(* IEC 61131-3 sources: moqui-plc/iec61131/moqui/framework/src/main/org/moqui/context, 20 files *)

(* ---- LogCmd.dut ---- *)
(*#-#-#-#-#-#-#-#-#-#---Declaration---#-#-#-#-#-#-#-#-#-#-#-#-#*)

{attribute 'qualified_only'}
TYPE LogCmd : (
    Idle := 0, (* Waiting for commands *)
    Push, (* Inserting a new log entry *)
	IncrementLast, (* Update the last log entry *)
	Peek, (* Read a log entry without removing it *)
	Pop, (* It actually removes the appended log entries *)
    Clear (* Complete buffer reset *)
); END_TYPE

(* ---- LogCmd.st ---- *)
TYPE LogCmd : (
    Idle := 0, (* Waiting for commands *)
    Push, (* Inserting a new log entry *)
	IncrementLast, (* Update the last log entry *)
	Peek, (* Read a log entry without removing it *)
	Pop, (* It actually removes the appended log entries *)
    Clear (* Complete buffer reset *)
); END_TYPE

(* ---- LogEvent.dut ---- *)
(*#-#-#-#-#-#-#-#-#-#---Declaration---#-#-#-#-#-#-#-#-#-#-#-#-#*)

TYPE LogEvent : STRUCT
	(* Unique identifier for the log event *)
    logEventId : STRING;
    loggerName : STRING;
	marker : LogMarker;
    level : LogLevel;
    logEventDate : DATE_AND_TIME;
	source : STRING;
	payloadType : LogPayloadType;
    payload : LogPayload;
	(* contextData: STRING; *)
	(* Number of times this log event was repeated, for compression *)
    repeatCount : UINT;
END_STRUCT END_TYPE

(* ---- LogEvent.st ---- *)
TYPE LogEvent : STRUCT
	(* Unique identifier for the log event *)
    logEventId : STRING;
    loggerName : STRING;
	marker : LogMarker;
    level : LogLevel;
    logEventDate : DATE_AND_TIME;
	source : STRING;
	payloadType : LogPayloadType;
    payload : LogPayload;
	(* contextData: STRING; *)
	(* Number of times this log event was repeated, for compression *)
    repeatCount : UINT;
END_STRUCT END_TYPE

(* ---- LogLevel.dut ---- *)
(*#-#-#-#-#-#-#-#-#-#---Declaration---#-#-#-#-#-#-#-#-#-#-#-#-#*)

{attribute 'qualified_only'}
TYPE LogLevel : (
	Trace := 0,
	Debug,
	Info,
	Warn,
	Error,
	Fatal,
	All,
	Off
); END_TYPE

(* ---- LogLevel.st ---- *)
TYPE LogLevel : (
	Trace := 0,
	Debug,
	Info,
	Warn,
	Error,
	Fatal,
	All,
	Off
); END_TYPE

(* ---- LogMarker.dut ---- *)
(*#-#-#-#-#-#-#-#-#-#---Declaration---#-#-#-#-#-#-#-#-#-#-#-#-#*)

{attribute 'qualified_only'}
{attribute 'strict'}
TYPE LogMarker : (
	Diagnostics := 0,
	Lifecycle,
	Integration,
	Health,
	Telemetry,
	AuditLog,
	Kpi,
	Measurement
); END_TYPE

(* ---- LogMarker.st ---- *)
TYPE LogMarker : (
	Diagnostics := 0,
	Lifecycle,
	Integration,
	Health,
	Telemetry,
	AuditLog,
	Kpi,
	Measurement
); END_TYPE

(* ---- LogPayload.dut ---- *)
(*#-#-#-#-#-#-#-#-#-#---Declaration---#-#-#-#-#-#-#-#-#-#-#-#-#*)

TYPE LogPayload : UNION
	message : STRING;
    enumValue : UINT;
    numericValue : LREAL;
END_UNION END_TYPE

(* ---- LogPayload.st ---- *)
TYPE LogPayload : UNION
	message : STRING;
    enumValue : UINT;
    numericValue : LREAL;
END_UNION END_TYPE

(* ---- LogPayloadType.dut ---- *)
(*#-#-#-#-#-#-#-#-#-#---Declaration---#-#-#-#-#-#-#-#-#-#-#-#-#*)

{attribute 'qualified_only'}
TYPE LogPayloadType : (
    Text := 0,
	Numeric,
	Enum
); END_TYPE

(* ---- LogPayloadType.st ---- *)
TYPE LogPayloadType : (
    Text := 0,
	Numeric,
	Enum
); END_TYPE

(* ---- LogSource.dut ---- *)
(*#-#-#-#-#-#-#-#-#-#---Declaration---#-#-#-#-#-#-#-#-#-#-#-#-#*)

TYPE LogSource : STRUCT
	(* Reference to log ring buffer *)
    logRef : REFERENCE TO LogRingBuffer;
	lastLogSize : UINT;
	lastHead : UINT := 1;
	lastTail : UINT := 1;
	lastOverflowCount : UDINT;
END_STRUCT END_TYPE

(* ---- LogSource.st ---- *)
TYPE LogSource : STRUCT
	(* Reference to log ring buffer *)
    logRef : REFERENCE TO LogRingBuffer;
	lastLogSize : UINT;
	lastHead : UINT := 1;
	lastTail : UINT := 1;
	lastOverflowCount : UDINT;
END_STRUCT END_TYPE

(* ---- ec.gvl ---- *)
(*#-#-#-#-#-#-#-#-#-#---Declaration---#-#-#-#-#-#-#-#-#-#-#-#-#*)

(* Execution Context *)
VAR_GLOBAL
    (* Timing generation *)
    clks : Clocks;

	(*
	 * Framework args.
	 * External framework commands and configurations set by Moqui or supervision.
     *)
	enable : BOOL := TRUE;
	init : BOOL := TRUE; (* It could be the powerOn signal*)
	fault, error, commError, reset, autoReset : BOOL;
	(* All device configs loaded *)
	allConfigLoaded : BOOL;
	retryCount, retryTime : UINT;
	isPrimary : BOOL;
	heartbeat : ULINT;

	(* Logger *)
    (* Array of reference to local logs used by the log appender *)
    logSourceList : ARRAY[1..LOG_SOURCE_LIST_MAX_SIZE] OF LogSource;
    logSourceListSize : UINT := 0;

	(* Facade for managing devices and logical parameters. *)
	dev : DeviceFacade;

	(* Facade for managing physical devices and input/output signals *)
	io : IOFacade;

	(* Optional: Moqui WorkEffort entity used for tracking information related to the execution of a production run. *)
	workEffort : WorkEffort;

	(* MQTT pub/sub commands *)
	connectionFactory : MqttConnectionFactory;
	logAppenderEnable : BOOL := TRUE;
	paramsPubEnable : BOOL := TRUE;
	paramsSubEnable : BOOL := TRUE;
END_VAR

(* ---- ec.st ---- *)
(* Execution Context *)
VAR_GLOBAL
    (* Timing generation *)
    clks : Clocks;

	(*
	 * Framework args.
	 * External framework commands and configurations set by Moqui or supervision.
     *)
	enable : BOOL := TRUE;
	init : BOOL := TRUE; (* It could be the powerOn signal*)
	fault, error, commError, reset, autoReset : BOOL;
	(* All device configs loaded *)
	allConfigLoaded : BOOL;
	retryCount, retryTime : UINT;
	isPrimary : BOOL;
	heartbeat : ULINT;

	(* Logger *)

    (* Array of reference to local logs used by the log appender *)
    logSourceList : ARRAY[1..LOG_SOURCE_LIST_MAX_SIZE] OF LogSource;
    logSourceListSize : UINT := 0;

	(* Facade for managing devices and logical parameters. *)
	dev : DeviceFacade;

	(* Facade for managing physical devices and input/output signals *)
	io : IOFacade;

	(* Optional: Moqui WorkEffort entity used for tracking information related to the execution of a production run. *)
	workEffort : WorkEffort;

	(* MQTT pub/sub commands *)
	connectionFactory : MqttConnectionFactory;
	logAppenderEnable : BOOL := TRUE;
	paramsPubEnable : BOOL := TRUE;
	paramsSubEnable : BOOL := TRUE;

	(* Motion override — written by Moqui via liveParamsSub *)
	trjDynamicSlowdownEnable : BOOL := FALSE;
	trjDynamicSlowdownFactor : LREAL := 1.0;
END_VAR

(* ---- LoggerFacade.pou ---- *)
(*#-#-#-#-#-#-#-#-#-#---Declaration---#-#-#-#-#-#-#-#-#-#-#-#-#*)

{attribute 'no_assign'}
(*
 * Logger with local circular buffer and duplicate suppression.
 * Designed for central orchestration by a global LogAppender.
 *)
FUNCTION_BLOCK LoggerFacade
VAR_EXTERNAL CONSTANT
	defaultLogLevel : LogLevel;
	LOG_SOURCE_LIST_MAX_SIZE : UINT;
END_VAR
VAR_EXTERNAL
	logSourceList : ARRAY[1..LOG_SOURCE_LIST_MAX_SIZE] OF LogSource;
    logSourceListSize : UINT;
END_VAR
(* Log event data *)
VAR_INPUT
    (* Trigger for logging a new event *)
    enable : BOOL;
	(*
     * Unique identifier for the log event.
     * If empty a UUID will be generated internally.
     *)
    logEventId : STRING := '';
    loggerName : STRING;
    level : LogLevel := defaultLogLevel;
	marker : LogMarker := LogMarker.Diagnostics;
	source : STRING;
    payloadType : LogPayloadType := LogPayloadType.Text;
	message : STRING;
    enumValue : UINT;
    numericValue : LREAL;
	(* contextData : STRING; (* Uncomment if needed *) *)
END_VAR
(* Configuration parameters *)
VAR_INPUT
	(* Duplicate suppression for log compression *)
	suppressDuplicates : BOOL := TRUE;
    (* Duplicate suppression window *)
    suppressDuration : TIME := T#10s;
END_VAR
VAR_OUTPUT
	done, error : BOOL;
END_VAR
VAR
	(* Local log ring buffer *)
    logBuffer : LogRingBuffer;
    init : BOOL := FALSE;
    isDuplicate : BOOL;
    now : DATE_AND_TIME;
    lastLogEvent : LogEvent;
	(* Log event ID generator *)
    timestamp : SysTimeRtc.SYSTIME;
    uuid : STRING(40);
END_VAR

(*#-#-#-#-#-#-#-#-#-#---Implementation---#-#-#-#-#-#-#-#-#-#-#-#-#*)

(* Register once into the log appender source list *)
IF NOT init THEN
    IF logSourceListSize < LOG_SOURCE_LIST_MAX_SIZE THEN
        logSourceListSize := logSourceListSize + 1;
        logSourceList[logSourceListSize].logRef REF= logBuffer;
    ELSE
        error := TRUE;
    END_IF;

    init := TRUE;
END_IF;

IF NOT enable THEN RETURN; END_IF;

now := nowTimestamp();
isDuplicate := FALSE;

(* Compression logic (duplicate suppression) *)
IF suppressDuplicates AND (payloadType = lastLogEvent.payloadType)
        AND (loggerName = lastLogEvent.loggerName)
		AND (source = lastLogEvent.loggerName) THEN
	CASE payloadType OF
		LogPayloadType.Text: isDuplicate := (message = lastLogEvent.payload.message);
		LogPayloadType.Enum: isDuplicate := (enumValue = lastLogEvent.payload.enumValue);
		LogPayloadType.Numeric: isDuplicate := (numericValue = lastLogEvent.payload.numericValue);
	END_CASE;
END_IF;

IF isDuplicate AND ((now - lastLogEvent.logEventDate) < suppressDuration) THEN
	(* Increment repeat counter instead of storing new entry *)
	logBuffer.cmd := LogCmd.IncrementLast;
ELSE
	(* Prepare the new log event entry *)
	IF logEventId = '' THEN
		SysTimeRtcHighResGet(pTimestamp := timestamp);
		uuid := CONCAT(loggerName, '-');
		uuid := CONCAT(uuid, ULINT_TO_STRING(timestamp));
		lastLogEvent.logEventId := uuid;
	ELSE
		lastLogEvent.logEventId := logEventId;
	END_IF;

	lastLogEvent.loggerName := loggerName;
	lastLogEvent.level := level;
	lastLogEvent.marker := marker;
	lastLogEvent.logEventDate := now;
	lastLogEvent.source := source;
	lastLogEvent.payloadType := payloadType;
	lastLogEvent.repeatCount := 1;
	(* lastLogEvent.contextData := contextData; *)

	CASE payloadType OF
		LogPayloadType.Text : lastLogEvent.payload.message := message;
		LogPayloadType.Enum : lastLogEvent.payload.enumValue := enumValue;
		LogPayloadType.Numeric: lastLogEvent.payload.numericValue := numericValue;
	END_CASE;

	(* Append the new log event *)
	logBuffer.logEntry := lastLogEvent;
	logBuffer.cmd := LogCmd.Push;
END_IF;

(* Execute local buffer operation *)
logBuffer();
logBuffer.cmd := LogCmd.Idle;

done := logBuffer.done;
error := error OR logBuffer.error;

(* ---- LoggerFacade.st ---- *)
(*
 * Logger with local circular buffer and duplicate suppression.
 * Designed for central orchestration by a global LogAppender.
 *)
FUNCTION_BLOCK LoggerFacade
	VAR_EXTERNAL CONSTANT
		defaultLogLevel : LogLevel;
		defaultLogSuppressDuration : TIME;
		defaultLogSuppressDuplicates : BOOL;
		LOG_SOURCE_LIST_MAX_SIZE : UINT;
	END_VAR
	VAR_EXTERNAL
		logSourceList : ARRAY[1..LOG_SOURCE_LIST_MAX_SIZE] OF LogSource;
	    logSourceListSize : UINT;
	END_VAR
	(* Log event data *)
	VAR_INPUT
	    (* Trigger for logging a new event *)
	    enable : BOOL;
		(*
	     * Unique identifier for the log event.
	     * If empty a UUID will be generated internally.
	     *)
	    logEventId : STRING := '';
	    loggerName : STRING;
	    level : LogLevel := defaultLogLevel;
		marker : LogMarker := LogMarker.Diagnostics;
		source : STRING;
	    payloadType : LogPayloadType := LogPayloadType.Text;
		message : STRING;
	    enumValue : UINT;
	    numericValue : LREAL;
		(* contextData : STRING; (* Uncomment if needed *) *)
	END_VAR
	(* Configuration parameters *)
	VAR_INPUT
		(* Duplicate suppression for log compression *)
		suppressDuplicates : BOOL := defaultLogSuppressDuplicates;
	    (* Duplicate suppression window *)
	    suppressDuration : TIME := defaultLogSuppressDuration;
	END_VAR
	VAR_OUTPUT
		done, error : BOOL;
	END_VAR
	VAR
		(* Local log ring buffer *)
	    logBuffer : LogRingBuffer;
	    init : BOOL := FALSE;
	    isDuplicate : BOOL;
	    now : DATE_AND_TIME;
	    lastLogEvent : LogEvent;
		(* Log event ID generator *)
	    timestamp : SysTimeRtc.SYSTIME;
	    uuid : STRING(40);
	END_VAR

	(* Register once into the log appender source list *)
	IF NOT init THEN
	    IF logSourceListSize < LOG_SOURCE_LIST_MAX_SIZE THEN
	        logSourceListSize := logSourceListSize + 1;
	        logSourceList[logSourceListSize].logRef REF= logBuffer;
	    ELSE
	        error := TRUE;
	    END_IF;

	    init := TRUE;
	END_IF;

	IF NOT enable THEN RETURN; END_IF;

	now := nowTimestamp();
	isDuplicate := FALSE;

	(* Compression logic (duplicate suppression) *)
	IF suppressDuplicates AND (payloadType = lastLogEvent.payloadType)
	        AND (loggerName = lastLogEvent.loggerName)
			AND (source = lastLogEvent.source) THEN
		CASE payloadType OF
			LogPayloadType.Text: isDuplicate := (message = lastLogEvent.payload.message);
			LogPayloadType.Enum: isDuplicate := (enumValue = lastLogEvent.payload.enumValue);
			LogPayloadType.Numeric: isDuplicate := (numericValue = lastLogEvent.payload.numericValue);
		END_CASE;
	END_IF;

	IF isDuplicate AND ((now - lastLogEvent.logEventDate) < suppressDuration) THEN
		(* Increment repeat counter instead of storing new entry *)
		logBuffer.cmd := LogCmd.IncrementLast;
	ELSE
		(* Prepare the new log event entry *)
		IF logEventId = '' THEN
			SysTimeRtcHighResGet(pTimestamp := timestamp);
			uuid := CONCAT(loggerName, '-');
			uuid := CONCAT(uuid, ULINT_TO_STRING(timestamp));
			lastLogEvent.logEventId := uuid;
		ELSE
			lastLogEvent.logEventId := logEventId;
		END_IF;

		lastLogEvent.loggerName := loggerName;
		lastLogEvent.level := level;
		lastLogEvent.marker := marker;
		lastLogEvent.logEventDate := now;
		lastLogEvent.source := source;
		lastLogEvent.payloadType := payloadType;
		lastLogEvent.repeatCount := 1;
		(* lastLogEvent.contextData := contextData; *)

		CASE payloadType OF
			LogPayloadType.Text : lastLogEvent.payload.message := message;
			LogPayloadType.Enum : lastLogEvent.payload.enumValue := enumValue;
			LogPayloadType.Numeric: lastLogEvent.payload.numericValue := numericValue;
		END_CASE;

		(* Append the new log event *)
		logBuffer.logEntry := lastLogEvent;
		logBuffer.cmd := LogCmd.Push;
	END_IF;

	(* Execute local buffer operation *)
	logBuffer();
	logBuffer.cmd := LogCmd.Idle;

	done := logBuffer.done;
	error := error OR logBuffer.error;
	END_FUNCTION_BLOCK

(* ---- LogRingBuffer.pou ---- *)
(*#-#-#-#-#-#-#-#-#-#---Declaration---#-#-#-#-#-#-#-#-#-#-#-#-#*)

{attribute 'no_assign'}
FUNCTION_BLOCK LogRingBuffer
VAR_EXTERNAL CONSTANT
    LOG_MAX_SIZE : UINT;
END_VAR
VAR_INPUT
    cmd : LogCmd := LogCmd.Idle;
    logEntry : LogEvent;
END_VAR
VAR_OUTPUT
    done, error, isFull, isEmpty : BOOL;
    head, tail : UINT := 1;
    (* Peek/Pop result: set on LogCmd.Peek and LogCmd.Pop *)
    headEntry : LogEvent;
    (* Exposed so that it can be cloned by the log appender (memcpy one-cycle operation). *)
    logBuffer : ARRAY[1..LOG_MAX_SIZE] OF LogEvent;
    logSize : UINT;
    overflowCount : UDINT;
END_VAR
VAR CONSTANT
	MAX_UDINT : UDINT := 16#FFFFFFFF;
END_VAR
VAR
    lastCommand : LogCmd := LogCmd.Idle;
    i : UINT;
END_VAR

(*#-#-#-#-#-#-#-#-#-#---Implementation---#-#-#-#-#-#-#-#-#-#-#-#-#*)

(* Reset instant outputs *)
done := FALSE;
error := FALSE;

(* Invariants guard *)
IF (head < 1) OR (head > LOG_MAX_SIZE) OR (tail < 1) OR (tail > LOG_MAX_SIZE) OR (logSize > LOG_MAX_SIZE) THEN
    head := 1; tail := 1; logSize := 0;
    error := TRUE;
    RETURN;
END_IF;

IF (overflowCount = MAX_UDINT) THEN overflowCount := 1; END_IF;

IF (cmd <> LogCmd.Idle) THEN
    CASE cmd OF
        LogCmd.Push :
            logBuffer[tail] := logEntry;

            IF (logSize >= LOG_MAX_SIZE) THEN
                (* Buffer full, overwrite oldest entries *)
                head := (head MOD LOG_MAX_SIZE) + 1;
                overflowCount := overflowCount + 1;
            ELSE
                logSize := logSize + 1;
            END_IF;

            tail := (tail MOD LOG_MAX_SIZE) + 1;
            done := TRUE;

        (* Increment repeat counter instead of storing new log entry *)
        LogCmd.IncrementLast :
            IF logSize = 0 THEN
				error := TRUE;
			ELSE
                i := tail - 1;
                IF i < 1 THEN i := LOG_MAX_SIZE; END_IF;

                (* Saturate repeatCount *)
                IF logBuffer[i].repeatCount < 65535 THEN
                    logBuffer[i].repeatCount := logBuffer[i].repeatCount + 1;
                END_IF;

				done := TRUE;
            END_IF;

        (* Returns head entry without removing it. Error if empty (Java Queue.peek semantics). *)
        LogCmd.Peek :
            IF logSize = 0 THEN
                error := TRUE;
            ELSE
                headEntry := logBuffer[head];
                done := TRUE;
            END_IF;

        (* Returns and removes head entry. Error if empty (Java Deque.pop semantics). *)
        LogCmd.Pop :
            IF logSize = 0 THEN
                error := TRUE;
            ELSE
                headEntry := logBuffer[head];
                head := (head MOD LOG_MAX_SIZE) + 1;
                logSize := logSize - 1;
                done := TRUE;
            END_IF;

        LogCmd.Clear :
            head := 1; tail := 1; logSize := 0; overflowCount := 0;
            done := TRUE;
    END_CASE;
END_IF;

lastCommand := cmd;
isEmpty := (logSize = 0);
isFull := (logSize = LOG_MAX_SIZE);

(* ---- LogRingBuffer.st ---- *)
FUNCTION_BLOCK LogRingBuffer
	VAR_EXTERNAL CONSTANT
	    LOG_MAX_SIZE : UINT;
	END_VAR
	VAR_INPUT
	    cmd : LogCmd := LogCmd.Idle;
	    logEntry : LogEvent;
	END_VAR
	VAR_OUTPUT
	    done, error, isFull, isEmpty : BOOL;
	    head, tail : UINT := 1;
	    (* Peek/Pop result: set on LogCmd.Peek and LogCmd.Pop *)
	    headEntry : LogEvent;
	    (* Exposed so that it can be cloned by the log appender (memcpy one-cycle operation). *)
	    logBuffer : ARRAY[1..LOG_MAX_SIZE] OF LogEvent;
	    logSize : UINT;
	    overflowCount : UDINT;
	END_VAR
	VAR CONSTANT
		MAX_UDINT : UDINT := 16#FFFFFFFF;
	END_VAR
	VAR
	    lastCommand : LogCmd := LogCmd.Idle;
	    i : UINT;
	END_VAR

	(* Reset instant outputs *)
	done := FALSE;
	error := FALSE;

	(* Invariants guard *)
	IF (head < 1) OR (head > LOG_MAX_SIZE) OR (tail < 1) OR (tail > LOG_MAX_SIZE) OR (logSize > LOG_MAX_SIZE) THEN
	    head := 1; tail := 1; logSize := 0;
	    error := TRUE;
	    RETURN;
	END_IF;

	IF (overflowCount = MAX_UDINT) THEN overflowCount := 1; END_IF;

	IF (cmd <> LogCmd.Idle) THEN
	    CASE cmd OF
	        LogCmd.Push :
	            logBuffer[tail] := logEntry;

	            IF (logSize >= LOG_MAX_SIZE) THEN
	                (* Buffer full, overwrite oldest entries *)
	                head := (head MOD LOG_MAX_SIZE) + 1;
	                overflowCount := overflowCount + 1;
	            ELSE
	                logSize := logSize + 1;
	            END_IF;

	            tail := (tail MOD LOG_MAX_SIZE) + 1;
	            done := TRUE;

	        (* Increment repeat counter instead of storing new log entry *)
	        LogCmd.IncrementLast :
	            IF logSize = 0 THEN
					error := TRUE;
				ELSE
	                i := tail - 1;
	                IF i < 1 THEN i := LOG_MAX_SIZE; END_IF;

	                (* Saturate repeatCount *)
	                IF logBuffer[i].repeatCount < 65535 THEN
	                    logBuffer[i].repeatCount := logBuffer[i].repeatCount + 1;
	                END_IF;

					done := TRUE;
	            END_IF;

	        (* Returns head entry without removing it. Error if empty (Java Queue.peek semantics). *)
	        LogCmd.Peek :
	            IF logSize = 0 THEN
	                error := TRUE;
	            ELSE
	                headEntry := logBuffer[head];
	                done := TRUE;
	            END_IF;

	        (* Returns and removes head entry. Error if empty (Java Deque.pop semantics). *)
	        LogCmd.Pop :
	            IF logSize = 0 THEN
	                error := TRUE;
	            ELSE
	                headEntry := logBuffer[head];
	                head := (head MOD LOG_MAX_SIZE) + 1;
	                logSize := logSize - 1;
	                done := TRUE;
	            END_IF;

	        LogCmd.Clear :
	            head := 1; tail := 1; logSize := 0; overflowCount := 0;
	            done := TRUE;
	    END_CASE;
	END_IF;

	lastCommand := cmd;
	isEmpty := (logSize = 0);
	isFull := (logSize = LOG_MAX_SIZE);
	END_FUNCTION_BLOCK
